Universal Robots PolyScope program: 30-seek_destack.urp

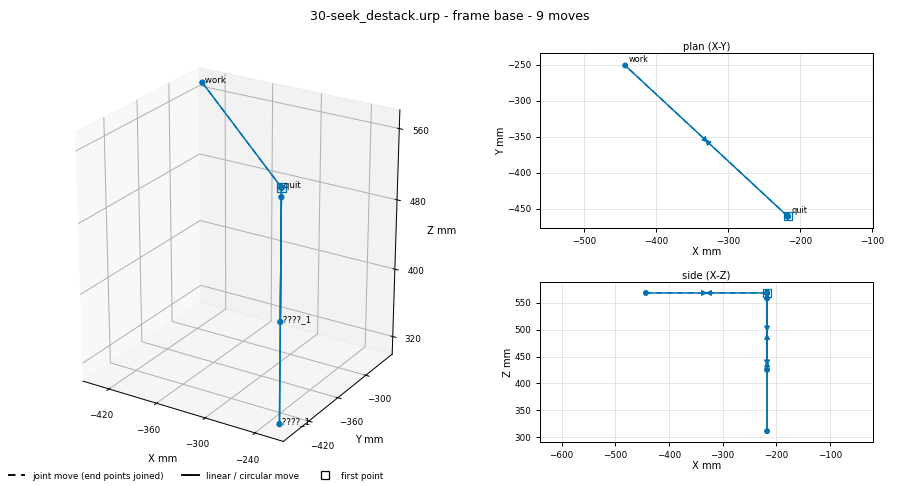
[picture p0: tool path of 30-seek_destack.urp in frame base, 9 of 9 moves have a stored position in this frame; points joined in program order, loops and branches not executed]
ProgramRoot directory=/home/ur/ursim-3.1/programs/basic training/30-seek_destack; kinematics=(a=[0.00021, -0.33281, -0.36715, -0.0002, 0.00018, 0], d=[0.08931, 141.17378, -190.60291, 49.5398, 0.09517, 0.08271], alpha=[1.57042, 0.00187, -0.00281, 1.57, -1.57028, 0], deltaTheta=[0.00006, 0.6718, -0.31, -0.36174, -0.00002, -0.00005], status=linearised); lastSavedInVersion=(project__name=Polyscope, major__version=3, minor__version=1, svn__revision=17195, build__date=Mar 11 2015, 13:02:28); name=30-seek_destack; programVersion=(project__name=Polyscope, major__version=3, minor__version=1, svn__revision=17141, build__date=Mar 06 2015, 07:52:30); robotEnvironmentFileName=default; serialNumberRobot=2014350001
  BeforeStart description=COMMAND_SEQUENCE_BEFORE_PROGRAM_START; name=BeforeStart
    Move cartesianAcceleration=1.2; cartesianSpeed=0.25; jointAcceleration=1.3962634015954636; jointSpeed=1.0471975511965976; sharedProcessMoveBlendRadius=0.025; motionType=CARTESIAN_SPACE
      Waypoint blendRadius=0.05; cartesianAcceleration=1.2; cartesianSpeed=0.25; jointAcceleration=1.3962634015954636; jointSpeed=1.0471975511965976; nextMotionTime=2.0; stoppoint=true; useSharedBlendParameter=true; useSharedParameters=true; outputFlangePose=(pos=(x=-0.21719219786801014, y=-0.46036716385432425, z=0.5685143889192367), rot=(x=0.9598588610265234, y=2.937589594293112, z=-0.003747393056620383)); position=TCP in base x=-217.182 y=-460.364 z=568.501 mm, rx=0.9599 ry=2.9376 rz=-0.0036 rad; joints [51.799, -85.253, 64.484, -68.326, -87.309, -2.059] deg; positionType=FIXED_POSITION; waypointPoseInFeatureCoordinates=(pos=(x=-0.21718230708247246, y=-0.4603641758056536, z=0.568501305188725), rot=(x=0.9598579128598694, y=2.9376437838387406, z=-0.0036385468739141063)); name=quit
  MainProgram cartesianAcceleration=1.2; cartesianSpeed=0.25; jointAcceleration=1.3962634015954636; jointSpeed=1.0471975511965976; sharedProcessMoveBlendRadius=0.025; motionType=JOINT_SPACE
    Stack cartesianAcceleration=1.2; cartesianSpeed=0.25; jointAcceleration=1.3962634015954636; jointSpeed=1.0471975511965976; sharedProcessMoveBlendRadius=0.025; motionType=CARTESIAN_SPACE; itemThikness=0.05; actionSequence=(MotionDefiningNode=(default=(cartesianAcceleration=1.2, cartesianSpeed=0.25, jointAcceleration=1.3962634015954636, jointSpeed=1.0471975511965976, recalculateMotions=false, sharedProcessMoveBlendRadius=0.025, motionType=CARTESIAN_SPACE)), AnchoredSequenceNode=(default=(name=拾取序列))); expr=ExpressionIONode≟ False; startPoint=(PositionNode=(default=(blendRadius=0.05, cartesianAcceleration=1.2, cartesianSpeed=0.25, jointAcceleration=1.3962634015954636, jointSpeed=1.0471975511965976, nextMotionTime=2.0, specifyNextMotionTime=false, stoppoint=true, useSharedBlendParameter=true, useSharedParameters=true, positionType=FIXED_POSITION)), WaypointNode=(default=(name=起始位置_1, relativeFromJointPositionVector=(joint=[nan, nan, nan, nan, nan, nan], isUndefined=true), relativeFromToolAxisAngle=(x=0.0, y=0.0, z=0.0), relativeFromToolPosition=(x=0.0, y=0.0, z=0.0)))); type=DESTACK
      Waypoint blendRadius=0.05; cartesianAcceleration=1.2; cartesianSpeed=0.25; jointAcceleration=1.3962634015954636; jointSpeed=1.0471975511965976; nextMotionTime=2.0; stoppoint=true; useSharedBlendParameter=true; useSharedParameters=true; outputFlangePose=(pos=(x=-0.21717619988589623, y=-0.46036921669142, z=0.42531105679832865), rot=(x=0.9597268187365741, y=2.937639793030738, z=-0.0038291905791459665)); position=TCP in base x=-217.17 y=-460.35 z=425.321 mm, rx=0.9597 ry=2.9376 rz=-0.0039 rad; joints [51.835, -88.698, 89.479, -89.876, -87.302, -2.091] deg; positionType=FIXED_POSITION; waypointPoseInFeatureCoordinates=(pos=(x=-0.21717037597705233, y=-0.4603501616740764, z=0.4253205809176114), rot=(x=0.9596681648311696, y=2.9376356621735074, z=-0.0038660732475922655)); name=起始位置_1
      Direction cartesianAcceleration=1.2; cartesianSpeed=0.01; jointAcceleration=1.3962634015954636; jointSpeed=1.0471975511965976; sharedProcessMoveBlendRadius=0.025; motionType=CARTESIAN_SPACE; maxDistance=-0.5; stopAtDistance=true; variable=0.0
        Waypoint blendRadius=0.05; cartesianAcceleration=1.2; cartesianSpeed=0.25; jointAcceleration=1.3962634015954636; jointSpeed=1.0471975511965976; nextMotionTime=2.0; stoppoint=true; useSharedBlendParameter=true; useSharedParameters=true; outputFlangePose=(pos=(x=-0.21714778413401273, y=-0.46037929998942956, z=0.5585273756889697), rot=(x=0.9596461033307022, y=2.9376757400758065, z=-0.003845769599808408)); position=TCP in base x=-217.183 y=-460.369 z=558.526 mm, rx=0.9597 ry=2.9377 rz=-0.0039 rad; joints [51.807, -85.761, 66.59, -69.927, -87.309, -2.064] deg; positionType=FIXED_POSITION; waypointPoseInFeatureCoordinates=(pos=(x=-0.2171826806421643, y=-0.46036941339924886, z=0.5585264251243057), rot=(x=0.9596720259700784, y=2.9376504636753284, z=-0.0038558726051131703)); name=源位置_1
        Waypoint blendRadius=0.05; cartesianAcceleration=1.2; cartesianSpeed=0.25; jointAcceleration=1.3962634015954636; jointSpeed=1.0471975511965976; nextMotionTime=2.0; stoppoint=true; useSharedBlendParameter=true; useSharedParameters=true; outputFlangePose=(pos=(x=-0.21714774603431636, y=-0.4603792513959683, z=0.3109088284274395), rot=(x=0.9596461024255464, y=2.937675740585791, z=-0.0038457694654958153)); position=TCP in base x=-217.153 y=-460.366 z=310.886 mm, rx=0.9597 ry=2.9376 rz=-0.0037 rad; joints [51.852, -86.223, 103.851, -106.724, -87.276, -2.116] deg; positionType=FIXED_POSITION; waypointPoseInFeatureCoordinates=(pos=(x=-0.21715263537404114, y=-0.4603664352481359, z=0.3108858171636456), rot=(x=0.9596811460425333, y=2.937622458170777, z=-0.003728949236540786)); name=目标位置_1
      AnchoredSequence cartesianAcceleration=1.2; cartesianSpeed=0.25; jointAcceleration=1.3962634015954636; jointSpeed=1.0471975511965976; sharedProcessMoveBlendRadius=0.025; motionType=CARTESIAN_SPACE; anchoredWaypointNode=(PositionNode=(default=(blendRadius=0.05, cartesianAcceleration=1.2, cartesianSpeed=0.25, jointAcceleration=1.3962634015954636, jointSpeed=1.0471975511965976, nextMotionTime=2.0, specifyNextMotionTime=false, stoppoint=true, useSharedBlendParameter=true, useSharedParameters=true, positionType=FIXED_POSITION)), WaypointNode=(default=(name=退出, relativeFromJointPositionVector=(joint=[nan, nan, nan, nan, nan, nan], isUndefined=true), relativeFromToolAxisAngle=(x=0.0, y=0.0, z=0.0), relativeFromToolPosition=(x=0.0, y=0.0, z=0.0)))); name=拾取序列
        Waypoint blendRadius=0.05; cartesianAcceleration=1.2; cartesianSpeed=0.25; jointAcceleration=1.3962634015954636; jointSpeed=1.0471975511965976; nextMotionTime=2.0; stoppoint=true; useSharedBlendParameter=true; useSharedParameters=true; outputFlangePose=(pos=(x=-0.21717612678323245, y=-0.4603691240386742, z=0.568529576857277), rot=(x=0.9597268190603994, y=2.9376397937608885, z=-0.003829190125762048)); position=TCP in base x=-217.192 y=-460.367 z=568.514 mm, rx=0.9599 ry=2.9376 rz=-0.0037 rad; joints [51.801, -85.254, 64.483, -68.327, -87.308, -2.062] deg; positionType=FIXED_POSITION; waypointPoseInFeatureCoordinates=(pos=(x=-0.21719219786806124, y=-0.46036716385432647, z=0.5685143894182176), rot=(x=0.9598588609438276, y=2.937589594319922, z=-0.00374739302213559)); name=堆垛位置_1
        Set 
        Wait 
        Waypoint blendRadius=0.05; cartesianAcceleration=1.2; cartesianSpeed=0.25; jointAcceleration=1.3962634015954636; jointSpeed=1.0471975511965976; nextMotionTime=2.0; stoppoint=true; useSharedBlendParameter=true; useSharedParameters=true; outputFlangePose=(pos=(x=-0.21717612678323245, y=-0.4603691240386742, z=0.568529576857277), rot=(x=0.9597268190603994, y=2.9376397937608885, z=-0.003829190125762048)); position=TCP in base x=-217.183 y=-460.366 z=568.527 mm, rx=0.9596 ry=2.9377 rz=-0.0038 rad; joints [51.801, -85.254, 64.483, -68.327, -87.308, -2.062] deg; positionType=FIXED_POSITION; waypointPoseInFeatureCoordinates=(pos=(x=-0.21718261066990785, y=-0.4603661837720865, z=0.5685270108106596), rot=(x=0.9596472496666375, y=2.9376601665677695, z=-0.003811040739459232)); name=退出
    Move cartesianAcceleration=1.2; cartesianSpeed=0.25; jointAcceleration=1.3962634015954636; jointSpeed=1.0471975511965976; sharedProcessMoveBlendRadius=0.025; motionType=CARTESIAN_SPACE
      Waypoint blendRadius=0.05; cartesianAcceleration=1.2; cartesianSpeed=0.25; jointAcceleration=1.3962634015954636; jointSpeed=1.0471975511965976; nextMotionTime=2.0; stoppoint=true; useSharedBlendParameter=true; useSharedParameters=true; outputFlangePose=(pos=(x=-0.21719219786801014, y=-0.46036716385432425, z=0.5685143889192367), rot=(x=0.9598588610265234, y=2.937589594293112, z=-0.003747393056620383)); position=TCP in base x=-217.182 y=-460.364 z=568.501 mm, rx=0.9599 ry=2.9376 rz=-0.0036 rad; joints [51.799, -85.253, 64.484, -68.326, -87.309, -2.059] deg; positionType=FIXED_POSITION; waypointPoseInFeatureCoordinates=(pos=(x=-0.21718230708247246, y=-0.4603641758056536, z=0.568501305188725), rot=(x=0.9598579128598694, y=2.9376437838387406, z=-0.0036385468739141063)); name=quit
    Move cartesianAcceleration=1.2; cartesianSpeed=0.25; jointAcceleration=1.3962634015954636; jointSpeed=1.0471975511965976; sharedProcessMoveBlendRadius=0.025; motionType=JOINT_SPACE
      Waypoint blendRadius=0.05; cartesianAcceleration=1.2; cartesianSpeed=0.25; jointAcceleration=1.3962634015954636; jointSpeed=1.0471975511965976; nextMotionTime=2.0; stoppoint=true; useSharedBlendParameter=true; useSharedParameters=true; outputFlangePose=(pos=(x=-0.4429139443593031, y=-0.2508737018145271, z=0.5685143889820217), rot=(x=1.8052538827571194, y=2.512058532990084, z=-0.027516929668133773)); position=TCP in base x=-442.931 y=-250.877 z=568.504 mm, rx=1.8054 ry=2.5121 rz=-0.0275 rad; joints [16.584, -85.253, 64.484, -68.326, -87.309, -2.059] deg; positionType=FIXED_POSITION; waypointPoseInFeatureCoordinates=(pos=(x=-0.44293127638240326, y=-0.2508766740091713, z=0.5685035899957657), rot=(x=1.8053609104375923, y=2.5120669225611842, z=-0.027502438543735293)); name=work
      Set 
    Move cartesianAcceleration=1.2; cartesianSpeed=0.25; jointAcceleration=1.3962634015954636; jointSpeed=1.0471975511965976; sharedProcessMoveBlendRadius=0.025; motionType=CARTESIAN_SPACE
      Waypoint blendRadius=0.05; cartesianAcceleration=1.2; cartesianSpeed=0.25; jointAcceleration=1.3962634015954636; jointSpeed=1.0471975511965976; nextMotionTime=2.0; stoppoint=true; useSharedBlendParameter=true; useSharedParameters=true; outputFlangePose=(pos=(x=-0.21719219786801014, y=-0.46036716385432425, z=0.5685143889192367), rot=(x=0.9598588610265234, y=2.937589594293112, z=-0.003747393056620383)); position=TCP in base x=-217.182 y=-460.364 z=568.501 mm, rx=0.9599 ry=2.9376 rz=-0.0036 rad; joints [51.799, -85.253, 64.484, -68.326, -87.309, -2.059] deg; positionType=FIXED_POSITION; waypointPoseInFeatureCoordinates=(pos=(x=-0.21718230708247246, y=-0.4603641758056536, z=0.568501305188725), rot=(x=0.9598579128598694, y=2.9376437838387406, z=-0.0036385468739141063)); name=quit
